Fanuc KAREL source: kt00869.KL

-- PROVISIONAL review KL for V770-1; original PC SHA256 859af2c86881da32474839773a3bcc76a401ff18cb69fef785db89fe1ef76a69
-- Incomplete behavior may be omitted. Consult companion uncertainty JSON. Do not deploy.
PROGRAM KT00869
%NOLOCKGROUP
VAR
  I1 : INTEGER
  I2 : INTEGER
  OUT : REAL
BEGIN
  -- UNRESOLVED_PC offsets 5-16; opcodes 2E,23
  -- UNRESOLVED_PC offsets 21-32; opcodes 2E,23
  -- UNRESOLVED_PC offsets 37-48; opcodes 2E,23
  -- UNRESOLVED_PC offsets 53-64; opcodes 2E,23
  -- UNRESOLVED_PC offsets 69-87; opcodes 27,27,21,64,76,64,23
  -- UNRESOLVED_PC offsets 92-96; opcodes 7F
END KT00869
